// TwinCAT 3 PLC project Sequencer
// ProgramVersion: 3.1.4024.0
// libraries:
//   Tc2_Standard, * (Beckhoff Automation GmbH)
//   Tc2_System, * (Beckhoff Automation GmbH)
//   Tc3_Module, * (Beckhoff Automation GmbH)
// project tree:
//   DUTs/ E_FlapState.TcDUT, ST_FlapControl.TcDUT (not stored)
//   DUTs/MainSupervisorStructures/RouteSelectionStructures/ ST_RouteStatus.TcDUT (not stored)
//   DUTs/MainSupervisorEnums/ E_AutoPhase.TcDUT (not stored), E_MainMode.TcDUT (not stored), E_MainOperation.TcDUT, E_MainState.TcDUT
//   DUTs/MainSupervisorEnums/RouteSelectionEnums/ E_Route.TcDUT (not stored)
//   DUTs/MainSupervisorStructures/ ST_DeviceDiag.TcDUT (not stored), ST_OperationsCmd.TcDUT (not stored), ST_ProcessCmd.TcDUT (not stored), ST_ProcessDiag.TcDUT, ST_ProcessStatus.TcDUT, ST_ProcessValues.TcDUT (not stored)
//   DUTs/OperationsEnums/BigBagFillingEnums/ E_BigBagFillingState.TcDUT (not stored), E_BigBagFillMode.TcDUT
//   DUTs/OperationsEnums/DischargeStateEnums/ E_DischargeState.TcTLEO
//   DUTs/OperationStructures/ ST_BigBagCmd.TcDUT, ST_BigBagMassBalanceStatus.TcDUT (not stored), ST_BigBagValues.TcDUT (not stored), ST_DischargeCmd.TcDUT, ST_BigBagDischargeStatus.TcDUT (not stored)
//   GVLs/ GVL.TcGVL (not stored)
//   / PlcTask.TcTTO (not stored)
//   POUs/FB/MainProcessSupervisor/Diagnostics/ FB_DeviceDiagnostics.TcPOU, FB_ProcessDiagnostics.TcPOU (not stored)
//   POUs/FB/MainProcessSupervisor/ FB_MainProcessSupervisor.TcPOU (not stored)
//   POUs/FB/MainProcessSupervisor/Services/ FB_RouteManager.TcPOU (not stored)
//   POUs/FB/Operations/DischargeR01ToVR01/ FB_DischargeR01ToVR01.TcPOU (not stored)
//   POUs/FB/ProcessModules/ FB_AirExtraction.TcPOU (not stored), FB_BigBagDischarge.TcPOU, FB_BigBagFilling.TcPOU (not stored), FB_BigBagMassBalance.TcPOU, FB_CaptureWeight.TcPOU (not stored), FB_MineralDosing.TcPOU (not stored), FB_MixingVR01.TcPOU, FB_SludgeDosing.TcPOU (not stored)
//   POUs/Function/ F_CalcWeightDelta.TcPOU (not stored)
//   POUs/ MAIN.TcPOU (not stored)
//   POUs/Processes/ DewateringProcess.TcPOU
// real-time tasks:
//   TASK PlcTask: cycle T#10ms, priority 20, ADS port 350

// ---- DUTs/E_FlapState.TcDUT
TYPE E_FlapState :
(
    IdleClosed := 0,
    Opening    := 10,
    Opened     := 20,
    Closing    := 30,
    Fault      := 90   // 🔥 nowy stan
);
END_TYPE

// ---- DUTs/MainSupervisorEnums/E_MainOperation.TcDUT
{attribute 'qualified_only'}
{attribute 'strict'}
TYPE E_MainOperation :
(
	NONE			:=	0,
	SBR_TO_R01		:=	1,
	R01_TO_VR01		:=	2,
	SBR_TO_WIATA	:=	3,
	R01_TO_WIATA	:=	4
);
END_TYPE

// ---- DUTs/MainSupervisorEnums/E_MainState.TcDUT
{attribute 'qualified_only'}
{attribute 'strict'}
TYPE E_MainState :
(
	RUN		:=	0,
	STOP	:=	1,
	PAUSE	:=	2,
	FAULT	:=	3
);
END_TYPE

// ---- DUTs/MainSupervisorStructures/ST_ProcessDiag.TcDUT
TYPE ST_ProcessDiag :
STRUCT
    bSPD01Fault              	  : BOOL;

    bPauseRequiredByProcess       : BOOL;
    bPauseNoLime                  : BOOL;
    bPauseNoPerlite               : BOOL;

    bSystemReady				  : BOOL;
END_STRUCT
END_TYPE

// ---- DUTs/MainSupervisorStructures/ST_ProcessStatus.TcDUT
TYPE ST_ProcessStatus :
STRUCT
    eMode                      : E_MainMode;
    eState                     : E_MainState;
    eOperation                 : E_MainOperation;
    eAutoPhase                 : E_AutoPhase;
	
	eAutoRouteReq				: E_Route;

    bAutoCycleActive           : BOOL;
    bManualCycleActive         : BOOL;

    bReadyToStart              : BOOL;
    bInPause                   : BOOL;
    bInFault                   : BOOL;

    iStatusCode                : INT;
END_STRUCT
END_TYPE

// ---- DUTs/OperationsEnums/BigBagFillingEnums/E_BigBagFillMode.TcDUT
{attribute 'qualified_only'}
{attribute 'strict'}
TYPE E_BigBagFillMode :
(
    BULK,       // wysyp szybki
    PRECISE     // wysyp precyzyjny
);
END_TYPE

// ---- DUTs/OperationsEnums/DischargeStateEnums/E_DischargeState.TcTLEO
{attribute 'qualified_only'}
{attribute 'strict'}
TYPE E_DischargeState :
(
    IDLE,                    // blok nieaktywny
    DOSE_SLUDGE,             // dozowanie osadu
    DOSE_PERLITE,            // dozowanie perlitu
    DOSE_LIME,               // dozowanie wapna
    MIXING,                  // mieszanie wsadu przed wysypem

    DISCHARGE_RUN,           // właściwy wysyp do Big Baga
    STOP_DRIVE_FOR_WEIGHING, // zatrzymanie napędu i zamykanie klapy przed ważeniem
    WAIT_SCALE_SETTLE,       // oczekiwanie na ustabilizowanie wagi
    EVALUATE_DISCHARGE,      // ocena efektu wysypu po stabilizacji wagi

    WAIT_BAG_CHANGE,         // oczekiwanie na wymianę worka
    DONE                     // zakończona operacja
);
END_TYPE

// ---- DUTs/OperationStructures/ST_BigBagCmd.TcDUT
TYPE ST_BigBagCmd :
STRUCT
    rBagActualMassManualSet  : REAL;  // wartość wpisana przez operatora
    bApplyBagActualMass      : BOOL;  // przycisk zatwierdzenia (monostabilny)
    bConfirmBagChange        : BOOL;  // potwierdzenie wymiany worka
END_STRUCT
END_TYPE

// ---- DUTs/OperationStructures/ST_DischargeCmd.TcDUT
TYPE ST_DischargeCmd :
STRUCT
    bEn_SludgeDosing   		: BOOL; // sterowanie blokiem dozowania osadu
    bEn_PerliteDosing  		: BOOL; // sterowanie blokiem dozowania perlitu
    bEn_LimeDosing     		: BOOL; // sterowanie blokiem dozowania wapna
    bEn_Mixing         		: BOOL; // sterowanie blokiem mieszania
    bEn_AirExtraction  		: BOOL; // sterowanie blokiem usuwania pyłu i pary
	bEn_BigBagDischarge		: BOOL; //sterowanie blokiem rozładunku do big bag
	bEn_BigBagMassBalance	: BOOL; // sterowanie blokiem bilansu masy w worku
END_STRUCT
END_TYPE

// ---- POUs/FB/MainProcessSupervisor/Diagnostics/FB_DeviceDiagnostics.TcPOU
FUNCTION_BLOCK FB_DeviceDiagnostics
VAR_INPUT
	    // Falownikowe
    bFault_SP02     		: BOOL;
    bCommOk_SP02    		: BOOL;
                    		
    bFault_M01      		: BOOL;
    bCommOk_M01     		: BOOL;
                    		
    bFault_M02      		: BOOL;
    bCommOk_M02     		: BOOL;
                    		
    bFault_M03      		: BOOL;
    bCommOk_M03     		: BOOL;
                    		
    // Bez falownika		
    bFault_BL01     		: BOOL;
    bFault_SC01     		: BOOL;
    bFault_SC02     		: BOOL;
    bFault_E01      		: BOOL;
    bFault_E02      		: BOOL;
	
END_VAR
VAR_OUTPUT
    bCriticalDeviceFault    : BOOL;

    bFault_Thermal          : BOOL;
    bFault_Comm             : BOOL;
    bFault_Inverter         : BOOL;

END_VAR
VAR
END_VAR

bFault_Comm :=
    (NOT bCommOk_SP02) OR
    (NOT bCommOk_M01)  OR
    (NOT bCommOk_M02)  OR
    (NOT bCommOk_M03);
	
bFault_Inverter :=
    bFault_SP02 OR
    bFault_M01  OR
    bFault_M02  OR
    bFault_M03;

bFault_Thermal :=
    bFault_BL01 OR
    bFault_SC01 OR
    bFault_SC02;
		

bCriticalDeviceFault :=
    bFault_Comm OR
    bFault_Inverter OR
    bFault_Thermal;

END_FUNCTION_BLOCK

// ---- POUs/FB/ProcessModules/FB_BigBagDischarge.TcPOU
FUNCTION_BLOCK FB_BigBagDischarge
VAR_INPUT
    bEnable                     : BOOL;     // aktywacja bloku wysypu do Big Baga

    rBagActualMass              : REAL;     // aktualna masa bieżącego worka przed rozpoczęciem wysypu
    rBagTargetMass_SP           : REAL;     // zadana masa aktualnego Big Baga

    rDosedBatchActual           : REAL;     // aktualna rzeczywista ilość zadozowana w cyklu rSludge + rLime +rPerlite
    rBatchDischargeToleranceKg  : REAL;     // tolerancja uznania, że bulk praktycznie cały już wyszedł

    rMassBeforeDischarge		: REAL;		// stabilna masa przed wysypem odczytana z wagi zawiera wsad z cyklu + zaleganie
	rActualWeight               : REAL;     // aktualna masa batch procesu odczytywana z wagi

    tBulkDischargeTime_SP       : TIME;     // maksymalny czas wysypu w trybie BULK

    uiFlapPosFast_SP            : UINT;     // pozycja klapy dla szybkiego wysypu
    uiFlapPosFine_SP            : UINT;     // pozycja klapy dla precyzyjnego wysypu
END_VAR

VAR_OUTPUT
    eFillMode                   : E_BigBagFillMode; // wybrany tryb wysypu

    uiFlapPosSp                 : UINT;     // zadana pozycja klapy 0..100%
    bDone                       : BOOL;     // zakończony etap wysypu
	
    rDischargedMassStep         : REAL;     // niestabilna masa zrzucona w aktualnym wysypie według bieżącego bilansu
    rMassMissingToBagTarget     : REAL;     // ile jeszcze brakuje do osiągnięcia targetu worka

    sDiag                       : T_MaxString; // komunikat diagnostyczny
END_VAR

VAR
    fbBulkTimer                 : TON;      // timer maksymalnego czasu wysypu bulk
	bEnablePrev                 : BOOL := FALSE; // poprzedni stan enable do wykrycia startu wysypu
	
END_VAR

// ---------------------------------------------------------
// DOMYŚLNE WYJŚCIA
// ---------------------------------------------------------
uiFlapPosSp := 0;          // domyślnie klapa zamknięta
bDone := FALSE;            // domyślnie etap wysypu nie jest zakończony
sDiag := '';               // domyślnie pusty komunikat


// ---------------------------------------------------------
// DETEKCJA STARTU NOWEGO WYSYPU
// ---------------------------------------------------------
IF bEnable AND NOT bEnablePrev THEN
    rMassMissingToBagTarget := rBagTargetMass_SP - rBagActualMass; // ile jeszcze brakuje do targetu worka

    IF rMassMissingToBagTarget < 0.0 THEN
        rMassMissingToBagTarget := 0.0; // zabezpieczenie przed wartością ujemną
    END_IF;

    // wybór trybu tylko raz, na starcie wysypu
    IF rDosedBatchActual <= rMassMissingToBagTarget THEN
        eFillMode := E_BigBagFillMode.BULK; // cały nowy wsad mieści się jeszcze do worka
    ELSE
        eFillMode := E_BigBagFillMode.PRECISE; // ten cykl może już domknąć worek
    END_IF;
END_IF;

bEnablePrev := bEnable;


// ---------------------------------------------------------
// BLOK NIEAKTYWNY
// ---------------------------------------------------------
IF NOT bEnable THEN
    fbBulkTimer(IN := FALSE, PT := tBulkDischargeTime_SP);
    uiFlapPosSp := 0;
    rDischargedMassStep := 0.0;
    sDiag := 'BigBagDischarge idle';
    RETURN;
END_IF;


// ---------------------------------------------------------
// OBLICZENIA BIEŻĄCE
// ---------------------------------------------------------
rDischargedMassStep := rMassBeforeDischarge - rActualWeight; // ile zeszło od ustalonej masy przed wysypem na biezaco
IF rDischargedMassStep < 0.0 THEN
    rDischargedMassStep := 0.0; // zabezpieczenie przed ujemną różnicą
END_IF;


// ---------------------------------------------------------
// LOGIKA TRYBÓW WYSYPU
// ---------------------------------------------------------
CASE eFillMode OF

    E_BigBagFillMode.BULK:
        sDiag := 'Wysyp bulk';
        uiFlapPosSp := uiFlapPosFast_SP; // szybki wysyp - klapa szeroko otwarta

        fbBulkTimer(IN := TRUE, PT := tBulkDischargeTime_SP);

        // zakończenie bulk:
        // 1) jeśli praktycznie cały nowy wsad już wyszedł
        // 2) albo jeśli minął maksymalny czas wysypu
        IF rDischargedMassStep >= (rDosedBatchActual - rBatchDischargeToleranceKg) THEN
            uiFlapPosSp := 0; // zamknij klapę
            fbBulkTimer(IN := FALSE, PT := tBulkDischargeTime_SP);
            bDone := TRUE;

        ELSIF fbBulkTimer.Q THEN
            uiFlapPosSp := 0; // zamknij klapę
            fbBulkTimer(IN := FALSE, PT := tBulkDischargeTime_SP);
            bDone := TRUE;
        END_IF;


    E_BigBagFillMode.PRECISE:
        sDiag := 'Wysyp precyzyjny';
        uiFlapPosSp := uiFlapPosFine_SP; // wolny / ostrożny wysyp
        fbBulkTimer(IN := FALSE, PT := tBulkDischargeTime_SP);

        // Na tym etapie nie robimy jeszcze finalnej oceny domknięcia worka z zakłóconej wagi.
        // Ten blok kończy tylko etap wysypu.
        // Na start przyjmujemy ten sam warunek masowy co dla batcha,
        // a właściwa ocena worka nastąpi później po zatrzymaniu napędu i stabilizacji wagi.
        IF rDischargedMassStep >= (rDosedBatchActual - rBatchDischargeToleranceKg) THEN
            uiFlapPosSp := 0; // zamknij klapę
            bDone := TRUE;
        END_IF;


ELSE
    uiFlapPosSp := 0;
    fbBulkTimer(IN := FALSE, PT := tBulkDischargeTime_SP);
END_CASE;

END_FUNCTION_BLOCK

// ---- POUs/FB/ProcessModules/FB_BigBagMassBalance.TcPOU
FUNCTION_BLOCK FB_BigBagMassBalance
VAR_INPUT
    bEnable                  : BOOL;
	
    rBagActualMass           : REAL;   // masa worka przed aktualnym cyklem
    rBagTargetMass_SP        : REAL;   // target worka   
	rMassBeforeDischarge	 : REAL;   // masa przed zrzutem stabilnie zważona	
    rMassAfterDischarge 	 : REAL;   // masa po zrzucie stabilnie zważona 	
	rBagFullToleranceKg      : REAL;   // tolerancja uznania worka za pełny
END_VAR
VAR_OUTPUT
    rBagActualMassNew        : REAL;   // nowa masa worka po aktualnym cyklu
    rMassToTarget            : REAL;   // ile brakuje do targetu
    bBagFull                 : BOOL;   // worek osiągnął target
    bBagChangeRequired       : BOOL;   // wymagana wymiana worka
    bDone                    : BOOL;
    sDiag                    : T_MaxString;
END_VAR
VAR
	rDischargeMass           : REAL;   // masa rzeczywiście zrzucona po stabilizacji
	bEnablePrev				 : BOOL:=FALSE;	//wejscie w pierwszy cykl
END_VAR

// domyślna diagnostyka
sDiag := 'BigBagMassBalance idle';

// obliczenie tylko raz na zboczu aktywacji
IF bEnable AND NOT bEnablePrev THEN

	// masa rzeczywiscie zrzucona na podstawie pomiarów stabilnych wagi
	rDischargeMass := rMassBeforeDischarge - rMassAfterDischarge; // Rzeczywista masa zrzutu       
    
	// nowa masa worka po aktualnym cyklu
    rBagActualMassNew := rBagActualMass + rDischargeMass;
 
    // ile jeszcze brakuje do targetu
    rMassToTarget := rBagTargetMass_SP - rBagActualMassNew;


    // ocena pełnego worka
    IF rBagActualMassNew >= (rBagTargetMass_SP - rBagFullToleranceKg) THEN
        bBagFull := TRUE;
        bBagChangeRequired := TRUE;
        sDiag := 'BigBag pelny - wymagana wymiana';
    ELSE
        bBagFull := FALSE;
        bBagChangeRequired := FALSE;
        sDiag := 'BigBag niepelny';
    END_IF;

    bDone := TRUE;
END_IF;

// reset gotowości po wyłączeniu enable
IF NOT bEnable THEN
    bDone := FALSE;
END_IF;

// pamięć poprzedniego stanu enable
bEnablePrev := bEnable;

END_FUNCTION_BLOCK

// ---- POUs/FB/ProcessModules/FB_MixingVR01.TcPOU
FUNCTION_BLOCK FB_MixingVR01
VAR_INPUT
	bEnable 	: BOOL; //uruchom mieszanie z zadaną czestotliwościa pracy
	rSpeedAuto	: REAL; //zadana częstotliwość pracy M01 i M02	
END_VAR
VAR_OUTPUT
	bCmd_M01	: BOOL;
	bCmd_M02    : BOOL;
	rSpeedSet	: REAL;
END_VAR

// ---------------------------------------------------------
// STOP GLOBALNY
// ---------------------------------------------------------
IF NOT bEnable THEN
	rSpeedAuto := 0.0;
	bCmd_M01 := FALSE;
	bCmd_M02 := FALSE;
ELSE
	rSpeedSet := rSpeedAuto;
	bCmd_M01 := TRUE;
	bCmd_M02 := TRUE;
END_IF

END_FUNCTION_BLOCK

// ---- POUs/Processes/DewateringProcess.TcPOU
PROGRAM DewateringProcess
VAR
	fbRouteManager			:	FB_RouteManager;
	fbProcessDiagnostics	:	FB_ProcessDiagnostics;
	fbDeviceDiagnostics		:	FB_DeviceDiagnostics;
	fbMainProcessSupervisor	:	FB_MainProcessSupervisor;
	
	fbDischargeR01ToVR01	:	FB_DischargeR01ToVR01;
	
	fbBigBagDischarge		:	FB_BigBagDischarge;
	fbBigBagMassBalance			:   FB_BigBagMassBalance;  			
	

END_VAR

ACT_DeviceDiagnostics();
ACT_ProcessDiagnostics();
ACT_RouteManager();
ACT_MainProcessSupervisor();

ACT_BigBagDischarge();
ACT_BigBagMassBalance();

//ACT_BigBagFilling();

ACTION ACT_BigBagDischarge:
GVL.g_stBigBagDischargeStatus.rDischargedMassStep := fbBigBagDischarge.rDischargedMassStep;
GVL.g_stBigBagDischargeStatus.uiFlapPosSp := fbBigBagDischarge.uiFlapPosSp;
GVL.g_stBigBagDischargeStatus.rMassMissingToBagTarget := fbBigBagDischarge.rMassMissingToBagTarget;
GVL.g_stBigBagDischargeStatus.sDiag := fbBigBagDischarge.sDiag;
fbBigBagDischarge(
    bEnable := GVL.g_stDischargeCmd.bEn_BigBagDischarge,
    rBagActualMass := GVL.g_stBigBagValues.rBagActualMass,
    rBagTargetMass_SP := 500,
    rDosedBatchActual := GVL.g_stBigBagValues.rDosedBatchActual,
    rBatchDischargeToleranceKg := 20,
    rMassBeforeDischarge := GVL.g_stBigBagValues.rMassBeforeDischarge,
    rActualWeight := GVL.g_rReactorActualMass,
    tBulkDischargeTime_SP := T#90s,
    uiFlapPosFast_SP := 90,
    uiFlapPosFine_SP := 30); // FB_BigBagDischarge
GVL.g_stBigBagDischargeStatus.eFillMode := fbBigBagDischarge.eFillMode;
GVL.g_stBigBagDischargeStatus.bDone := fbBigBagDischarge.bDone;
END_ACTION

ACTION ACT_BigBagFilling:
fbBigBagFilling(
    bEnable := GVL.g_Enable,
    bConfirmBagChange := GVL.g_bConfirmBagChange,
    bLoadStartBagMass := GVL.g_bLoadStartBagMass,
    rStartBagMass := GVL.g_rStartBagMass,
    rReactorActualMass := GVL.g_rReactorActualMass,
    rBagTargetMass_SP := 500,
    rBagToleranceKg := 10,
    rCycleMassActual := GVL.g_rCycleMassActual,
    rCycleDischargeToleranceKg := 10,
    tBulkDischargeTime_SP := T#60s,
    uiFlapPosFast_SP := 100,
    uiFlapPosFine_SP := 30); // FB_BigBagFilling
END_ACTION

ACTION ACT_BigBagMassBalance:
fbBigBagMassBalance(
    bEnable := GVL.g_stDischargeCmd.bEn_BigBagMassBalance,
    rBagActualMass := GVL.g_stBigBagValues.rBagActualMass,
    rBagTargetMass_SP := 450,
    rMassBeforeDischarge := GVL.g_stBigBagValues.rMassBeforeDischarge,
    rMassAfterDischarge := GVL.g_stBigBagValues.rMassAfterDischarge,
    rBagFullToleranceKg := 20); // FB_BigBagMassBalance
GVL.g_stBigBagMassbalanceStatus.rBagActualMassNew := fbBigBagMassBalance.rBagActualMassNew;
GVL.g_stBigBagMassbalanceStatus.rMassToTarget := fbBigBagMassBalance.rMassToTarget;
GVL.g_stBigBagMassbalanceStatus.bBagFull := fbBigBagMassBalance.bBagFull;
GVL.g_stBigBagMassbalanceStatus.bBagChangeRequired := fbBigBagMassBalance.bBagChangeRequired;
GVL.g_stBigBagMassbalanceStatus.bDone := fbBigBagMassBalance.bDone;
GVL.g_stBigBagMassbalanceStatus.sDiag := fbBigBagMassBalance.sDiag;
END_ACTION

ACTION ACT_DeviceDiagnostics:
GVL.g_stDeviceDiag.bFault_Thermal := fbDeviceDiagnostics.bFault_Thermal;
GVL.g_stDeviceDiag.bFault_Comm := fbDeviceDiagnostics.bFault_Comm;
GVL.g_stDeviceDiag.bFault_Inverter := fbDeviceDiagnostics.bFault_Inverter;
fbDeviceDiagnostics(
    bFault_SP02 := False,
    bCommOk_SP02 := True,
    bFault_M01 := False,
    bCommOk_M01 := True,
    bFault_M02 := False,
    bCommOk_M02 := True,
    bFault_M03 := False,
    bCommOk_M03 := True,
    bFault_BL01 := False,
    bFault_SC01 := False,
    bFault_SC02 := False,
    bFault_E01 := False,
    bFault_E02 := False); // FB_DeviceDiagnostics
GVL.g_stDeviceDiag.bCriticalDeviceFault := fbDeviceDiagnostics.bCriticalDeviceFault;
END_ACTION

ACTION ACT_MainProcessSupervisor:
fbMainProcessSupervisor(
    eModeCmd := GVL.g_stProcessCmd.eModeCmd,
    eManualOperationCmd := GVL.g_stProcessCmd.eManualOperationCmd,
    bCmdStartReq := GVL.g_stProcessCmd.bStartReq,
    bCmdPauseReq := GVL.g_stProcessCmd.bPauseReq,
    bCmdStopReq := GVL.g_stProcessCmd.bStopReq,
    eConfirmedRoute := GVL.g_stRouteStatus.eConfirmedRoute,
    bRouteValid := GVL.g_stRouteStatus.bRouteValid,
    bSystemReady := GVL.g_stProcessDiag.bSystemReady,
    bPauseRequiredByProcess := GVL.g_stProcessDiag.bPauseRequiredByProcess,
    bPauseNoLime := GVL.g_stProcessDiag.bPauseNoLime,
    bPauseNoPerlite := GVL.g_stProcessDiag.bPauseNoPerlite,
    bCriticalDeviceFault := GVL.g_stDeviceDiag.bCriticalDeviceFault,
    bSPD01FaultActive := GVL.g_stProcessDiag.bSPD01Fault,
    rR01Level := GVL.g_stProcessValues.rR01Level,
    rLevelMinSP := GVL.g_stProcessValues.rLevelMinSP,
    rLevelMaxSP := GVL.g_stProcessValues.rLevelMaxSP); // FB_MainProcessSupervisor
GVL.g_stProcessStatus.eState := fbMainProcessSupervisor.eState;
GVL.g_stProcessStatus.eOperation := fbMainProcessSupervisor.eOperation;
GVL.g_stProcessStatus.eAutoPhase := fbMainProcessSupervisor.eAutoPhase;
GVL.g_stProcessStatus.eAutoRouteReq := fbMainProcessSupervisor.eAutoRouteReq;
GVL.g_stProcessCmd.stOperationsCmd.bRunDischargeR01ToVR01 := fbMainProcessSupervisor.bCmdRunDischargeR01ToVR01;
GVL.g_stProcessCmd.stOperationsCmd.bRunFeedSBRtoR01 := fbMainProcessSupervisor.bCmdRunFeedSBRToR01;
GVL.g_stProcessCmd.stOperationsCmd.bRunSBRToWiata := fbMainProcessSupervisor.bCmdRunSBRToWiata;
GVL.g_stProcessCmd.stOperationsCmd.bRunR01ToWiata := fbMainProcessSupervisor.bCmdRunR01ToWiata;
GVL.g_stProcessStatus.iStatusCode := fbMainProcessSupervisor.iStatusCode;
GVL.g_stProcessStatus.bReadyToStart := fbMainProcessSupervisor.bReadyToStart;
END_ACTION

ACTION ACT_ProcessDiagnostics:
GVL.g_stProcessDiag.bPauseRequiredByProcess := fbProcessDiagnostics.bPauseRequiredByProcess;
GVL.g_stProcessDiag.bPauseNoLime := fbProcessDiagnostics.bPauseNoLime;
GVL.g_stProcessDiag.bPauseNoPerlite := fbProcessDiagnostics.bPauseNoPerlite;
fbProcessDiagnostics(
    bCriticalDeviceFault := GVL.g_stDeviceDiag.bCriticalDeviceFault,
    bLimeAvailable := True,
    bPerliteAvailable := True,
    bSPD01Fault := False); // FB_ProcessDiagnostics
GVL.g_stProcessDiag.bSPD01Fault := fbProcessDiagnostics.bSPD01FaultActive;
GVL.g_stProcessDiag.bSystemReady := fbProcessDiagnostics.bSystemReady;
END_ACTION

ACTION ACT_RouteManager:
fbRouteManager(
    eMode := GVL.g_stProcessCmd.eModeCmd,
    bConfirmRouteReq := GVL.g_stProcessCmd.bConfirmRouteReq,
    eSelectedRoute := GVL.g_stRouteStatus.eSelectedRoute,
    eAutoRouteReq := GVL.g_stProcessStatus.eAutoRouteReq); // FB_RouteManager
GVL.g_stRouteStatus.eConfirmedRoute := fbRouteManager.eConfirmedRoute;
GVL.g_stRouteStatus.bRouteValid := fbRouteManager.bRouteValid;
GVL.g_stRouteStatus.iState := fbRouteManager.iState;
END_ACTION

END_PROGRAM
